(* PLC project State Machine Example.project, CODESYS CODESYS V3.5 SP20 Patch 1 *)
(* stored: creationDateTime 2025-05-31T21:59:47.386968, modificationDateTime 2025-05-31T21:59:31.9410502 *)

{attribute 'contains_implicit_enum'}
PROGRAM Main
  VAR
    scanCount : INT;
    StateHandler : StateMachineHandler;
    {attribute 'implicit_enum_type'}
    state : Implicit_Enum__Main__state;
  END_VAR

                    
state := StateHandler.CurrentState;

CASE StateHandler.CurrentState OF
	
	Init: HandleInitState();
	
	Run: HandleRunState();
	
	Stop: HandleStopState();
	
	Error: HandleErrorState();
	
END_CASE

scanCount := scanCount+1;


                  

METHOD HandleInitState : BOOL
                          
IF scanCount >= 200 THEN
	scanCount := 0;
	StateHandler.UpdateState(Run);
END_IF
                        
END_METHOD

METHOD HandleRunState : BOOL
                          
IF scanCount >= 200 THEN
	scanCount := 0;
	StateHandler.UpdateState(Stop);
END_IF
                        
END_METHOD

METHOD HandleStopState : BOOL
                          
IF scanCount >= 200 THEN
	scanCount := 0;
	StateHandler.UpdateState(Init);
END_IF
                        
END_METHOD

METHOD HandleErrorState : BOOL
                          
                        
END_METHOD
END_PROGRAM

FUNCTION_BLOCK StateMachineHandler
  VAR
    _currentState : INT;
    _lastState : INT;
  END_VAR

                    
                  

METHOD UpdateState : BOOL
  VAR_INPUT
    requestedState : INT;
  END_VAR
                          
IF requestedState <> _currentState THEN
	_lastState := _currentState;
	_currentState := requestedState;
END_IF
                        
END_METHOD

PROPERTY CurrentState : INT
GET
                            
CurrentState := _currentState;
                          
END_GET
END_PROPERTY

PROPERTY LastState : INT
GET
                            
LastState := _lastState;
                          
END_GET
END_PROPERTY
END_FUNCTION_BLOCK

CONFIGURATION Device
  RESOURCE Application ON PLC
    TASK MainTask(INTERVAL := T#20ms, PRIORITY := 1);
    PROGRAM Main WITH MainTask : Main;
  END_RESOURCE
END_CONFIGURATION
